// TIA Portal project "Project2" (V16)

(* hardware
DEVICE "S7-1200 station_1"  S7-1200 Station
   slot 0: "Rack_0"  S7-1200 Rack  Rack  V1.0
   slot 1: "PLC Powered Off"  CPU 1214C AC/DC/Rly  6ES7 214-1BG40-0XB0  V4.2
*)

// ===== PLC "PLC Powered Off"  CPU 1214C AC/DC/Rly =====

VAR_GLOBAL   // PLC tag table "Default tag table"
   ""Start"" AT %I1.1 : Bool;
   ""Stop"" AT %I1.2 : Bool;
   ""M0"" AT %Q0.6 : Bool;
   ""M3"" AT %Q0.7 : Bool;
   ""M4"" AT %Q1.1 : Bool;
END_VAR